// TIA Portal V20 export
// export: Created 2025-12-01T14:57:12.1589021Z, ExportSetting None, DisplayName Totally Integrated Automation Portal, DisplayVersion V20 Update 3, DisplayName TIA Portal Openness, DisplayVersion V20 Update 3, DisplayName TIA Portal Version Control Interface, DisplayVersion V20 Update 3, DisplayName STEP 7 Professional, DisplayVersion V20 Update 3, DisplayName STEP 7 Safety, DisplayVersion V20 Update 2, DisplayName WinCC Basic/Comfort/Advanced, DisplayVersion V20 Update 3, DisplayName WinCC Professional, DisplayVersion V20 Update 3, DisplayName WinCC Unified, DisplayVersion V20 Update 3
FUNCTION "FC992_CTRL_VAR_Lenze_i550_Profinet" : Void   // FC992, STL
TITLE = Comunicación con variador Lenze Profinet
{ S7_Optimized_Access := 'FALSE' }
AUTHOR : VARIADOR
NAME : 20150506
VERSION : 3.2
// stored: AutoNumber false
   VAR_INPUT
      NumDispositivo : UInt;   // Numero dispositivo profinet
      DirInicial : UInt;   // Dirección inicio periferia
      Avance : Bool;
      Retroceso : Bool;
      Rearme : Bool;
      Homing : Bool;   // Solo para Elevadores ECO
      SentidoGiro : Bool;   // Cambia el sentido de giro
      Activar_DO1 : Bool;   // Al activar esta entrada, activamos la salida correspondiente XXXX.7 Ej: Dir INI 2000 - Q2000.7
      ConsignaVelocidad : UInt;   // Consigna en Hz
      Emergencia : Bool;   // Solo para Elevadores ECO
   END_VAR
   VAR_OUTPUT
      Freno : Bool;
   END_VAR
   VAR_TEMP
      EstadoVariador : Struct
         "Digital input 1" : Bool;
         "Digital input 2" : Bool;
         "Digital input 3" : Bool;
         "Digital input 4" : Bool;
         "Digital input 5" : Bool;
         Running : Bool;
         "Reserva 2" : Bool;
         "Reserva 3" : Bool;
         "Ready for operation" : Bool;
         "Auto setp active" : Bool;
         "Actual speed = 0" : Bool;
         Error : Bool;
         "Safe torque off" : Bool;
         "At current limit" : Bool;
         "At torque limit" : Bool;
         "Speed - set = act" : Bool;
      END_STRUCT;
      ControlVariador : Struct
         "Reserva 1" : Bool;
         "Reserva 2" : Bool;
         "Reserva 3" : Bool;
         "Reserva 4" : Bool;
         "Reserva 5" : Bool;
         "Reserva 6" : Bool;
         "Reserva 7" : Bool;
         "Salida Digital (DO1) = 1" : Bool;
         "Run forward" : Bool;
         "Reverse rotation dirtect." : Bool;
         "Reset error" : Bool;
         "Position counter reset" : Bool;
         "Activate quick stop" : Bool;
         "Sel. paramset b0" : Bool;
         "Sel. paramset b1" : Bool;
         "Reserva 11" : Bool;
      END_STRUCT;
      CodigoError : UInt;
      FrecuenciaActual : Int;
      CorrienteActual : Int;
      PosicionEncoder : Real;
      ACC : Int;
      DCC : Int;
      Termico_Tx : Int;
      P_EstadoVariador : DWord;
      P_ControlVariador : DWord;
      ReturnValor : Int;
      Cero : Byte;
   END_VAR
   VAR CONSTANT
      Constant_1 : Int;
   END_VAR
BEGIN

NETWORK
TITLE = Inicializar la temporales.
//////////////////////////////////////////////////////////////////////////////////////////
//////////////////////////////////////////////////////////////////////////////////////////
//////////////////////////////////////////////////////////////////////////////////////////
/// -- Inicializar las variables temporales
      L     P##EstadoVariador;
      T     #P_EstadoVariador;
      L     P##ControlVariador;
      T     #P_ControlVariador;

      L     0;
      T     LW [#P_EstadoVariador];
      T     LW [#P_ControlVariador];



NETWORK
TITLE = Lectura de Entradas del Variador
// En este segmeto leemos toda la inforamcion del Variador y lo guardamos en el DB 
// correspondiente
//////////////////////////////////////////////////////////////////////////////////////////
//////////////////////////////////////////////////////////////////////////////////////////
//////////////////////////////////////////////////////////////////////////////////////////
/// --- Leemos toda la inforamcion del Variador y lo guardamos en el DB correspondiente
      L     #DirInicial;  // Calculo puntero datos donde vamos a ir recogiendo la información
      SLD   3;
      LAR2;


//////////////////////////////////////////////////////////////////////////////////////////
//////////////////////////////////////////////////////////////////////////////////////////
//////////////////////////////////////////////////////////////////////////////////////////
/// --- Leemos todos los datos de periferia
      L     IW [AR2, P#0.0];  // Status word
      T     LW [#P_EstadoVariador];
      L     IW [AR2, P#2.0];  // Error Code
      T     #CodigoError;

      L     IW [AR2, P#4.0];  // Velocidad actual
      T     #FrecuenciaActual;
      L     IW [AR2, P#6.0];  // Corriente actual
      T     #CorrienteActual;

      L     ID [AR2, P#8.0];  // Posción motor actual (solo con encoder)
      DTR;
      L     65536.0;
      /R;
      T     #PosicionEncoder;


//////////////////////////////////////////////////////////////////////////////////////////
//////////////////////////////////////////////////////////////////////////////////////////
//////////////////////////////////////////////////////////////////////////////////////////
/// --- Guardamos datos recogidos del variador en la DB.

      CALL  MOVE
      ( IN  := #EstadoVariador,
        OUT := "DB940_Datos_VAR_Lenze_i550".Lenze_i550[#NumDispositivo]."Estatus variador"
      );

      L     #CodigoError;
      T     "DB940_Datos_VAR_Lenze_i550".Lenze_i550[#NumDispositivo]."Código de error";
      L     #FrecuenciaActual;
      T     "DB940_Datos_VAR_Lenze_i550".Lenze_i550[#NumDispositivo]."Frecuencia actual";
      L     #CorrienteActual;
      T     "DB940_Datos_VAR_Lenze_i550".Lenze_i550[#NumDispositivo]."Corriente actual";

      L     #PosicionEncoder;
      T     "DB940_Datos_VAR_Lenze_i550".Lenze_i550[#NumDispositivo]."Posicion encoder";

//////////////////////////////////////////////////////////////////////////////////////////
//////////////////////////////////////////////////////////////////////////////////////////
//////////////////////////////////////////////////////////////////////////////////////////
FinalLecturaVariador:NOP   0;



NETWORK
TITLE = Selección de juego de parámetros - PARA EL FUTURO
// Se deja preparado pero todo comentado. En el caso de que se usase hay que quitar los comentarios y añadir como Input de la funcion el bool "Motor_2"
//////////////////////////////////////////////////////////////////////////////////////////
//////////////////////////////////////////////////////////////////////////////////////////
//////////////////////////////////////////////////////////////////////////////////////////
//  Lenze tiene la opcion de poder controlar 4 tipos de variadores distintos.
//  Para proteger cada uno de ellos utilizamos la logica entre 2 bits.
//  Esta opción se denomina Parameter change-over en el software de Lenze (Easy starter)
//  Juego de parámetros 1 y 2 se van a utilizar para el control de 2 motores en triangulo
//  Juego de parámetros 3 y 4 se van a utilizar para el control de 2 motores en estrella.

//////////////////////////////////////////////////////////////////////////////////////////
//////////////////////////////////////////////////////////////////////////////////////////
//////////////////////////////////////////////////////////////////////////////////////////
// Seleccionar lista de parametros 1 // Triángulo MOTOR 1
//      SET
//      UN    #ConexionEstrella
//      UN    #Motor_2
//      SPBN  M2

//      R     #ControlVariador."Sel. paramset b0"
//      R     #ControlVariador."Sel. paramset b1"
//      SPA   MF

//////////////////////////////////////////////////////////////////////////////////////////
//////////////////////////////////////////////////////////////////////////////////////////
//////////////////////////////////////////////////////////////////////////////////////////
// Seleccionar lista de parametros 2 // Triángulo MOTOR 2
//M2:   SET
//      UN    #ConexionEstrella
//      U     #Motor_2
//      SPBN  M3
//      S     #ControlVariador."Sel. paramset b0"
//      R     #ControlVariador."Sel. paramset b1"

//      SPA   MF

//////////////////////////////////////////////////////////////////////////////////////////
//////////////////////////////////////////////////////////////////////////////////////////
//////////////////////////////////////////////////////////////////////////////////////////
// Seleccionar lista de parametros 3 // Estrella MOTOR 1
//M3:   SET
//      U     #ConexionEstrella
//      UN    #Motor_2
//      SPBN  M4
//      R     #ControlVariador."Sel. paramset b0"
//      S     #ControlVariador."Sel. paramset b1"

//      SPA   MF

//////////////////////////////////////////////////////////////////////////////////////////
//////////////////////////////////////////////////////////////////////////////////////////
//////////////////////////////////////////////////////////////////////////////////////////
// Seleccionar lista de parametros 4 //  Estrella MOTOR 2
//M4:   SET
//      U     #ConexionEstrella
//      U     #Motor_2
//      SPBN  MF
//      S     #ControlVariador."Sel. paramset b0"
//      S     #ControlVariador."Sel. paramset b1"

//////////////////////////////////////////////////////////////////////////////////////////
//////////////////////////////////////////////////////////////////////////////////////////
//////////////////////////////////////////////////////////////////////////////////////////
//MF:   NOP 0



NETWORK
TITLE = Rearme
//////////////////////////////////////////////////////////////////////////////////////////
//////////////////////////////////////////////////////////////////////////////////////////
//////////////////////////////////////////////////////////////////////////////////////////
// -- Enviar el rearme al variador
      SET;
      A     #Rearme;
      =     #ControlVariador."Reset error";



NETWORK
TITLE = Quick Stop
//////////////////////////////////////////////////////////////////////////////////////////
//////////////////////////////////////////////////////////////////////////////////////////
//////////////////////////////////////////////////////////////////////////////////////////
// -- Enviar el rearme al variador
      SET;
      AN    #Emergencia;
      =     #ControlVariador."Activate quick stop";



NETWORK
TITLE = Homing
//////////////////////////////////////////////////////////////////////////////////////////
//////////////////////////////////////////////////////////////////////////////////////////
//////////////////////////////////////////////////////////////////////////////////////////
// -- Enviar Homing (puesta a cero del encoder)
      SET;
      A     #Homing;
      =     #ControlVariador."Position counter reset";



NETWORK
TITLE = Estado DO1
//////////////////////////////////////////////////////////////////////////////////////////
//////////////////////////////////////////////////////////////////////////////////////////
//////////////////////////////////////////////////////////////////////////////////////////
// -- Enviar la salida digital DO1
      SET;
      A     #Activar_DO1;
      =     #ControlVariador."Salida Digital (DO1) = 1";



NETWORK
TITLE = Avance y Retroceso
// Para que todos los variadores tengan el mismo programa generamos un patilla de 
// sentido de giro para cambiar el sentido desde el PLC y mantener las entradas de 
// Avance y Retroceso
//////////////////////////////////////////////////////////////////////////////////////////
//////////////////////////////////////////////////////////////////////////////////////////
//////////////////////////////////////////////////////////////////////////////////////////
// -- Orden de avance
      SET;
      A(;
      O     #Avance;
      O     #Retroceso;
      );
      A     #EstadoVariador."Ready for operation";
      A     #EstadoVariador."Auto setp active";
      AN    #EstadoVariador."Safe torque off";
      AN    #EstadoVariador.Error;
      =     #ControlVariador."Run forward";



NETWORK
TITLE = Adaptación del Avance y Retroceso
// Para que todos los variadores tengan el mismo programa generamos un patilla de 
// sentido de giro para cambiar el sentido desde el PLC y mantener las entradas de 
// Avance y Retroceso
//////////////////////////////////////////////////////////////////////////////////////////
//////////////////////////////////////////////////////////////////////////////////////////
//////////////////////////////////////////////////////////////////////////////////////////
// Para que todos los variadores tengan el mismo programa generamos un patilla de
// sentido de giro para cambiar el sentido desde el PLC y mantener las entradas de
// Avance y Retroceso
//////////////////////////////////////////////////////////////////////////////////////////
//////////////////////////////////////////////////////////////////////////////////////////
//////////////////////////////////////////////////////////////////////////////////////////
      SET;
      A     #SentidoGiro;
      JC    SG;

      SET;
      A     #Retroceso;
      A     #EstadoVariador."Ready for operation";
      AN    #EstadoVariador."Safe torque off";
      AN    #EstadoVariador.Error;
      =     #ControlVariador."Reverse rotation dirtect.";
      JU    SF;

//////////////////////////////////////////////////////////////////////////////////////////
//////////////////////////////////////////////////////////////////////////////////////////
//////////////////////////////////////////////////////////////////////////////////////////
SG:   SET;
      A     #Avance;
      A     #EstadoVariador."Ready for operation";
      AN    #EstadoVariador."Safe torque off";
      AN    #EstadoVariador."Reserva 3";
      AN    #EstadoVariador.Error;
      =     #ControlVariador."Reverse rotation dirtect.";

//////////////////////////////////////////////////////////////////////////////////////////
//////////////////////////////////////////////////////////////////////////////////////////
//////////////////////////////////////////////////////////////////////////////////////////
SF:   NOP   0;



NETWORK
TITLE = Error de termico
// Señal para usar en el error de termico de la mesa
//////////////////////////////////////////////////////////////////////////////////////////
//////////////////////////////////////////////////////////////////////////////////////////
//////////////////////////////////////////////////////////////////////////////////////////
// -- Termico

      A     #EstadoVariador."Ready for operation";
      A     #EstadoVariador."Auto setp active";
      AN    #EstadoVariador."Safe torque off";
      AN    #EstadoVariador.Error;
      =     "DB940_Datos_VAR_Lenze_i550".Lenze_i550[#NumDispositivo].Termico_Tx;



NETWORK
TITLE = Activar Freno
// IMPORTANTE: Esta salida solo se usa para los elevadores ECO, porque tienen 2 frenos, uno que lo activa el variador y otro que lo activa el PLC con esta salida. En transporte no se usa esta salida poner una variable booleana Basura en su patilla de salida
/////////////////////////////////////////////////////////////////////////////////////////
//////////////////////////////////////////////////////////////////////////////////////////
//////////////////////////////////////////////////////////////////////////////////////////
/// --- SOLO PARA ELEVADORES ECO, EN TRANSPORTE NO SE USA
/// --- Recibimos del variador la confirmacion de que esta activando el Freno y usamos esa
/// --- confirmacion para activar el freno del armario
      A     "DB940_Datos_VAR_Lenze_i550".Lenze_i550[#NumDispositivo]."Estatus variador"."Release Holding Brake";
      =     #Freno;


NETWORK
TITLE = Escritura de las Salidas del Variador
//////////////////////////////////////////////////////////////////////////////////////////
//////////////////////////////////////////////////////////////////////////////////////////
//////////////////////////////////////////////////////////////////////////////////////////
/// --- Recoger datos a Enviar del Variador
      L     "DB940_Datos_VAR_Lenze_i550".Lenze_i550[#NumDispositivo].ACC;
      T     #ACC;
      L     "DB940_Datos_VAR_Lenze_i550".Lenze_i550[#NumDispositivo].DCC;
      T     #DCC;


//////////////////////////////////////////////////////////////////////////////////////////
//////////////////////////////////////////////////////////////////////////////////////////
//////////////////////////////////////////////////////////////////////////////////////////
/// --- Escribimos toda la inforamcion del Variador y lo guardamos en el DB correspondiente
      L     #DirInicial;  // Calculo puntero datos donde vamos a ir recogiendo la información
      SLD   3;
      LAR2;

      L     LW [#P_ControlVariador];  // Control Word
      T     QW [AR2, P#0.0];


// Consigna de velocidad
      L     #ConsignaVelocidad;
      T     QW [AR2, P#2.0];
      T     "DB940_Datos_VAR_Lenze_i550".Lenze_i550[#NumDispositivo]."Consigna de frecuencia";
// ACC
      L     #ACC;
      T     QW [AR2, P#4.0];
// DCC
      L     #DCC;
      T     QW [AR2, P#6.0];


//////////////////////////////////////////////////////////////////////////////////////////
//////////////////////////////////////////////////////////////////////////////////////////
//////////////////////////////////////////////////////////////////////////////////////////
/// Guardar en el DB
      CALL  MOVE
      ( IN  := #ControlVariador,
        OUT := "DB940_Datos_VAR_Lenze_i550".Lenze_i550[#NumDispositivo]."Palabra de control"
      );

      L     #ConsignaVelocidad;
      T     "DB940_Datos_VAR_Lenze_i550".Lenze_i550[#NumDispositivo]."Consigna de frecuencia";


END_FUNCTION
